// TIA Portal V17 export
// export: Created 2022-10-14T12:26:43.1758349Z, ExportSetting WithDefaults, DisplayName Totally Integrated Automation Portal, DisplayVersion V17 Update 4, DisplayName TIA Portal Openness, DisplayVersion V17 Update 4, DisplayName TIA Portal Version Control Interface, DisplayVersion V17, DisplayName SINAMICS Startdrive Advanced, DisplayVersion V17 Update2, DisplayName SINAMICS Startdrive G130, G150, S120, S150, SINAMICS MV, S210, DisplayVersion V17 Update2, DisplayName SINAMICS Startdrive G110M, G120, G120C, G120D, G120P, G115D, DisplayVersion V17 Update2, DisplayName STEP 7 Professional, DisplayVersion V17 Update 4, DisplayName STEP 7 Safety, DisplayVersion V17, DisplayName WinCC Advanced / Unified PC, DisplayVersion V17 Update 4
FUNCTION "1003_SEND_RECV" : Void   // FC1003, FBD
{ S7_Optimized_Access := 'TRUE' }
VERSION : 0.1
// stored: AutoNumber false, IsIECCheckEnabled false, SetENOAutomatically false, UDAEnableTagReadback false
   VAR_INPUT
      HW_RCV : HW_SUBMODULE;
      HW_SND : HW_SUBMODULE;
      "Message-Typ" : Byte;
      SubSysAdr : Byte;
      SND_ID : Byte;
      Adr : Byte;
      Kanal : Byte;
   END_VAR
   VAR_OUTPUT
      Error : Bool;
      RCV_ID : Byte;
      Data_RCV : "RCV_Dates";
   END_VAR
   VAR_TEMP
      H_DWord : DWord;
      RCV : Struct
         ID : Byte;
         "Messwert 1" : Byte;
         "Messwert 2" : Byte;
         "Messwert 3" : Byte;
         "Messwert 4" : Byte;
         Alarm : Byte;
         Einheit : Byte;
         "Beschreibung High" : Byte;
         "Beschreibung Low" : Byte;
         "Byte 9" : Byte;
      END_STRUCT;
      SND : Struct
         ID : Byte;
         "Message-Typ" : Byte;
         Subsystemadresse : Byte;
         Geräteadresse : Byte;
         Kanal : Byte;
         "Byte 5" : Byte;
         "Byte 6" : Byte;
         "Byte 7" : Byte;
         "Byte 8" : Byte;
         "Byte 9" : Byte;
         "Byte 10" : Byte;
      END_STRUCT;
      ERR1 : Int;
      ERR2 : Int;
   END_VAR
BEGIN

REGION Network 1: ####SEND####
END_REGION

REGION Network 2: Fortlaufende ID-Nr.
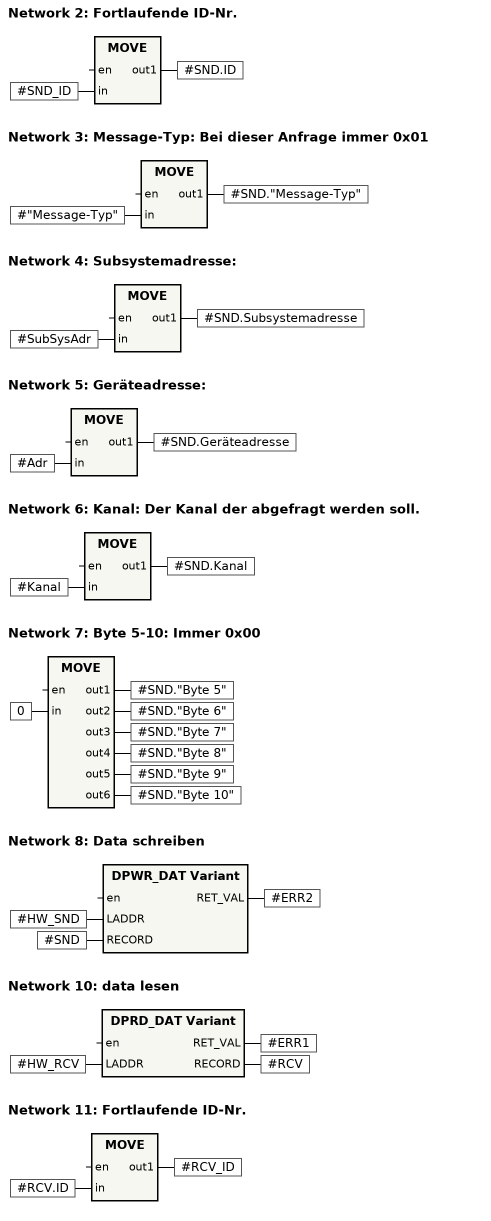
   #SND.ID := #SND_ID;
END_REGION

REGION Network 3: Message-Typ: Bei dieser Anfrage immer 0x01
   #SND."Message-Typ" := #"Message-Typ";
END_REGION

REGION Network 4: Subsystemadresse:
   // Je nachdem wie das Gerät betrieben wird, entweder die BCOM- oder
   // die externe BMS-Bus-Adresse (Default bei Einsatz im internen BMS-Bus: 2)
   #SND.Subsystemadresse := #SubSysAdr;
END_REGION

REGION Network 5: Geräteadresse:
   // Die interne BMS- oder BCOM-Adresse. Je nachdem, über welche Schnittstelle
   // das Gerät eingebunden ist.
   #SND.Geräteadresse := #Adr;
END_REGION

REGION Network 6: Kanal: Der Kanal der abgefragt werden soll.
   #SND.Kanal := #Kanal;
END_REGION

REGION Network 7: Byte 5-10: Immer 0x00
   #SND."Byte 5" := 0;
   #SND."Byte 6" := 0;
   #SND."Byte 7" := 0;
   #SND."Byte 8" := 0;
   #SND."Byte 9" := 0;
   #SND."Byte 10" := 0;
END_REGION

REGION Network 8: Data schreiben
   #ERR2 := DPWR_DAT(LADDR := #HW_SND, RECORD := #SND);
END_REGION

REGION Network 9: ####RECV####
END_REGION

REGION Network 10: data lesen
   #ERR1 := DPRD_DAT(LADDR := #HW_RCV, RECORD => #RCV);
END_REGION

REGION Network 11: Fortlaufende ID-Nr.
   #RCV_ID := #RCV.ID;
END_REGION

REGION Network 12: Byte 1-4: Messwerte
   // Die Daten werden als Float-Wert ausgegeben.
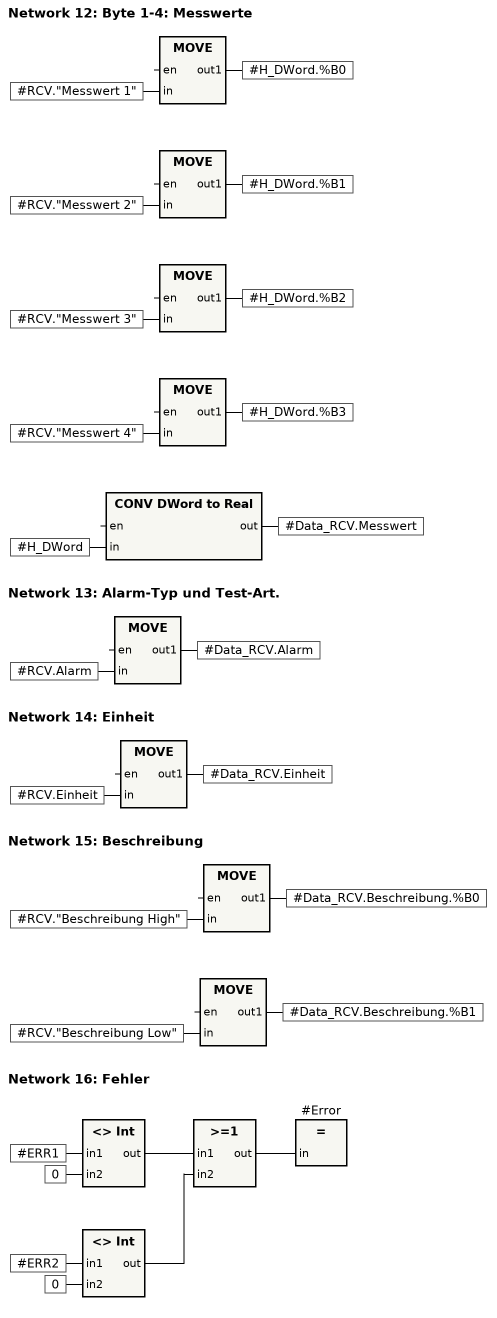
   #H_DWord.%B0 := #RCV."Messwert 1";
   #H_DWord.%B1 := #RCV."Messwert 2";
   #H_DWord.%B2 := #RCV."Messwert 3";
   #H_DWord.%B3 := #RCV."Messwert 4";
   #Data_RCV.Messwert := DWORD_TO_REAL(#H_DWord);
END_REGION

REGION Network 13: Alarm-Typ und Test-Art.
   // =============================================
   // Byte Bedeutung
   // Der Alarm-Typ ist durch die Bits 0 bis 2 codiert
   // Die Bits 3 und 4 sind reserviert und haben stets den Wert 0.
   // Bit 5 hat normalerweise den Wert 0 und steht für den digitalen Wert des Status
   // Diese Spalte ist nur für das SMI472 relevant.
   // Bit 6 oder 7 sind gesetzt, wenn ein interner oder externer Test abgelaufen ist.
   // Andere Werte sind reserviert.
   // Das komplette Byte wird aus der Summe von Alarm-Typ und Test-Art errechnet.
   // ____________________________________________________________________________________
   // 
   // Bit          7                        6                5                  4                    3                  2              1         0
   //        Test extern     Test intern     Status     Reserviert     Reserviert     Alarm     Fehler
   // _______________________________________________________________________________________
   // Alarm-Typ
   // Bit 7 6 5 4 3 2 1 0          Bedeutung
   //       X X X X X 0 0 0            Kein Alarm
   //       X X X X X 0 0 1            Vorwarnung
   //       0 0 X X X 0 1 0            Gerätefehler
   //       X X X X X 0 1 1            Reserviert
   //       X X X X X 1 0 0           Alarm (gelbe LED), z. B. Isolationsfehler
   //       X X X X X 1 0 1           Alarm (rote LED)
   //       X X X X X 1 1 0           Reserviert
   //       X X X X X … … …         Reserviert
   //       X X X X X 1 1 1          Reserviert
   // --------------------------------------------------------------------------------------------
   // Test
   // Bit 7 6 5 4 3 2 1 0          Bedeutung
   //      0 0 X X X X X X            Kein Test
   //      0 1 X X X X X X            Interner Test
   //      1 0 X X X X X X           Externer Test
   #Data_RCV.Alarm := #RCV.Alarm;
END_REGION

REGION Network 14: Einheit
   // Aufbau des Bytes: Bereich und Einheit.
   // ------------------------------------------------------------------------------------------------------
   // In den Bits 0 bis 4 ist die Einheit codiert.
   // Die Bits 6 und 7 beschreiben den Gültigkeitsbereich eines Werts.
   // ----------------------------------------------------------------------------------------------------------------------------------------------
   // Einheit
   // Bit 7 6 5 4 3 2 1 0          Bedeutung
   //       X X X 0 0 0 0 0         Ungültig (init)
   //       X X X 0 0 0 0 1         Keine Einheit
   //       X X X 0 0 0 1 0                Ω
   //       X X X 0 0 0 1 1                A
   //       X X X 0 0 1 0 0                V
   //       X X X 0 0 1 0 1                %
   //       X X X 0 0 1 1 0                Hz
   //       X X X 0 0 1 1 1             Baud
   //       X X X 0 1 0 0 0                 F
   //       X X X 0 1 0 0 1                H
   //       X X X 0 1 0 1 0                °C
   //       X X X 0 1 0 1 1                °F
   //       X X X 0 1 1 0 0            Sekunde
   //       X X X 0 1 1 0 1            Minute
   //       X X X 0 1 1 1 0           Stunde
   //       X X X 0 1 1 1 1           Tag
   //       X X X 1 0 0 0 0           Monat
   //       X X X … … … … …        Reserviert
   //       X X X 1 1 1 1 0            CODE
   //       X X X 1 1 1 1 1           Reserviert
   //       X X X … … … … …        Reserviert
   //       X X X 1 1 1 1 1           Reserviert
   // ----------------------------------------------------------------------------------
   // Gültigkeitsbereich
   // Bit 7 6 5 4 3 2 1 0     Bedeutung
   //       0 0 X X X X X X    Wahrer Wert
   //       0 1 X X X X X X    Wahrer Wert ist kleiner
   //       1 0 X X X X X X    Wahrer Wert ist größer
   //       1 1 X X X X X X    Ungültiger Wert
   #Data_RCV.Einheit := #RCV.Einheit;
END_REGION

REGION Network 15: Beschreibung
   // Beschreibung High: Das High-Byte der Messwert-Beschreibung.
   // Beschreibung Low: Das Low-Byte der Messwert Beschreibung.
   #Data_RCV.Beschreibung.%B0 := #RCV."Beschreibung High";
   #Data_RCV.Beschreibung.%B1 := #RCV."Beschreibung Low";
END_REGION

REGION Network 16: Fehler
   #Error := (#ERR1 <> 0) OR (#ERR2 <> 0);
END_REGION
END_FUNCTION
